# B&R Automation Studio project Mapp6D_Demo (part 2)

#### Variables.var - Local variables
```iecst
VAR
	DemoMacro : ARRAY[0..99] OF Macro_typ;
	gMacro : ARRAY[0..99] OF Macro_typ;
	MC_BR_MoveInPlaneAsync_Acp6D_0 : MC_BR_MoveInPlaneAsync_Acp6D;
	MC_BR_Move6D_Acp6D_0 : MC_BR_Move6D_Acp6D;
	MC_BR_MoveArc_Acp6D_0 : MC_BR_MoveArc_Acp6D;
	MC_BR_AsmPowerOn_Acp6D_0 : MC_BR_AsmPowerOn_Acp6D;
	MC_BR_MacroCreate_Acp6D_0 : MC_BR_MacroCreate_Acp6D;
	MC_BR_MoveInPlane_Acp6D_0 : MC_BR_MoveInPlane_Acp6D;
	MC_BR_AsmReadStatus_0 : MC_BR_AsmReadStatus_Acp6D;
	MC_BR_MacroSave_0 : MC_BR_MacroSave_Acp6D;
	MC_BR_MacroClear_0 : MC_BR_MacroClear_Acp6D;
	MC_BR_MacroDelete_0 : MC_BR_MacroDelete_Acp6D;
	MC_BR_MacroRun_0 : MC_BR_MacroRun_Acp6D;
	MC_BR_AsmGetShuttle_0 : MC_BR_AsmGetShuttle_Acp6D;
END_VAR
VAR CONSTANT
	MAX_NUM_SH : USINT := 10;
	C_MOVE_IN_PLANE_010 : USINT := 10;
	C_MOVE_IN_PLANE_ASYNC_015 : USINT := 15;
	C_MOVE_IN_6D_PLANE_020 : USINT := 20;
	C_MOVE_ARC_025 : USINT := 25;
	C_NEXT_COMMAND_05 : USINT := 5;
END_VAR
VAR
	Cmd : Ctrl_typ;
	i : USINT;
	inc : USINT;
	MacroState : USINT;
	visMacroStatus : STRING[80];
	MacroSh : {REDUND_UNREPLICABLE} ARRAY[0..9] OF Mc6DShuttleType;
	TempName : STRING[33];
	ExistingMacroNames : ARRAY[0..19] OF STRING[28];
	MacroName : STRING[28];
	helpStr : STRING[28];
	int_to_str : STRING[4];
	ShRefArr : ARRAY[0..MAX_NUM_SH] OF Mc6DShuttleType;
	macroLine : UDINT;
	command : UINT;
	Clear : BOOL;
	ReRun : BOOL;
	RunMacro : BOOL;
	CenterSegX : REAL;
	CenterSegY : REAL;
	SecondPosY : REAL;
	SecondPosX : REAL;
	FirstPosY : REAL;
	FirstPosX : REAL;
	visLockRun : BOOL;
	PathCW : McAcp6DInPlanePathEnum;
	PathACW : McAcp6DInPlanePathEnum;
END_VAR
VAR CONSTANT
	C_WAIT_00 : USINT := 0;
	C_READ_STATUS_01 : USINT := 1;
	C_POWER_ON_02 : USINT := 2;
	C_CREATE_03 : USINT := 3;
	C_DELETE_04 : USINT := 4;
	C_SAVE_60 : USINT := 60;
	C_REMAKE_DEMO_MACRO_70 : USINT := 70;
	C_RUN_DEMO_MACRO_80 : USINT := 80;
	C_RUN_DEMO_MACRO_81 : USINT := 81;
	C_RUN_DEMO_MACRO_82 : USINT := 82;
	C_RUN_DEMO_MACRO_83 : USINT := 83;
	C_RE_RUN_85 : USINT := 85;
	C_CLEARMACRO_90 : USINT := 90;
	C_RESET_100 : USINT := 100;
END_VAR
```

#### DemoAct.st
```iecst
ACTION DemoAct:

	// DEMO MACRO
	macroLine := 0;
	XY_MIN; 			// Min position on one segment 0.6 `
	XY_MAX; 			// Max position on one segment 0.240
	SEG_CENTER;			// Middle position 0.120

	// Calculate the min and max movement positions allowed

	IF inc = 0 THEN // System Top right 1st position
		FirstPosX := gAssemblyX_max;
		FirstPosY := gAssemblyY_max;
		SecondPosX := XY_MIN;
		SecondPosY := XY_MIN;
		CenterSegX := SEG_CENTER;
		CenterSegY := SEG_CENTER;
		PathCW := mcACP6D_PATH_Y_THEN_X;
		PathACW := mcACP6D_PATH_X_THEN_Y;
	ELSIF inc = 1 THEN // Bottom Left of system 1st position
		FirstPosX := XY_MIN;
		FirstPosY := XY_MIN;
		SecondPosX := gAssemblyX_max;
		SecondPosY := gAssemblyY_max;
		CenterSegX := gAssemblyX_max - HALF_SHUTTLE;
		CenterSegY := gAssemblyY_max - HALF_SHUTTLE;
		PathCW := mcACP6D_PATH_Y_THEN_X;
		PathACW := mcACP6D_PATH_X_THEN_Y;
	ELSIF inc = 2 THEN // Top left of system 1st position
		FirstPosX := XY_MIN;
		FirstPosY := gAssemblyY_max;
		SecondPosX := gAssemblyX_max;
		SecondPosY := XY_MIN;
		CenterSegX := gAssemblyX_max - HALF_SHUTTLE;
		CenterSegY := SEG_CENTER;
		PathCW := mcACP6D_PATH_X_THEN_Y;
		PathACW := mcACP6D_PATH_Y_THEN_X;
	ELSIF inc = 3 THEN // Bottom right of system 1st position
		FirstPosX := gAssemblyX_max;
		FirstPosY := XY_MIN;
		SecondPosX := XY_MIN;
		SecondPosY := gAssemblyY_max;
		CenterSegX := SEG_CENTER;
		CenterSegY := gAssemblyY_max - HALF_SHUTTLE;
		PathCW := mcACP6D_PATH_X_THEN_Y;
		PathACW := mcACP6D_PATH_Y_THEN_X;
	END_IF

	// Round edge twice total CWise

	DemoMacro[macroLine].ShuttleID := 1;
	DemoMacro[macroLine].CommandType := C_MOVE_IN_PLANE_010;
	DemoMacro[macroLine].MovePlane.Velocity := 2.0;
	DemoMacro[macroLine].MovePlane.Acceleration := 20.0;
	DemoMacro[macroLine].MovePlane.EndVelocity := 0.0;
	DemoMacro[macroLine].MovePlane.Position.X := FirstPosX;
	DemoMacro[macroLine].MovePlane.Position.Y := FirstPosY;
	DemoMacro[macroLine].MovePlane.Path := PathCW;

	macroLine := macroLine + 1;

	DemoMacro[macroLine].ShuttleID := 1;
	DemoMacro[macroLine].CommandType := C_MOVE_IN_PLANE_010;
	DemoMacro[macroLine].MovePlane.Velocity := 2.0;
	DemoMacro[macroLine].MovePlane.Acceleration := 20.0;
	DemoMacro[macroLine].MovePlane.EndVelocity := 0.0;
	DemoMacro[macroLine].MovePlane.Position.X := SecondPosX;
	DemoMacro[macroLine].MovePlane.Position.Y := SecondPosY;
	DemoMacro[macroLine].MovePlane.Path := PathCW;

	macroLine := macroLine + 1;

	DemoMacro[macroLine].ShuttleID := 1;
	DemoMacro[macroLine].CommandType := C_MOVE_IN_PLANE_010;
	DemoMacro[macroLine].MovePlane.Velocity := 2.0;
	DemoMacro[macroLine].MovePlane.Acceleration := 20.0;
	DemoMacro[macroLine].MovePlane.EndVelocity := 0.0;
	DemoMacro[macroLine].MovePlane.Position.X := FirstPosX;
	DemoMacro[macroLine].MovePlane.Position.Y := FirstPosY;
	DemoMacro[macroLine].MovePlane.Path := PathCW;

	macroLine := macroLine + 1;

	DemoMacro[macroLine].ShuttleID := 1;
	DemoMacro[macroLine].CommandType := C_MOVE_IN_PLANE_010;
	DemoMacro[macroLine].MovePlane.Velocity := 2.0;
	DemoMacro[macroLine].MovePlane.Acceleration := 20.0;
	DemoMacro[macroLine].MovePlane.EndVelocity := 0.0;
	DemoMacro[macroLine].MovePlane.Position.X := SecondPosX;
	DemoMacro[macroLine].MovePlane.Position.Y := SecondPosY;
	DemoMacro[macroLine].MovePlane.Path := PathCW;

	macroLine := macroLine + 1;

	// Move to center and dance...
	DemoMacro[macroLine].ShuttleID 					  := 1;
	DemoMacro[macroLine].CommandType 				  := C_MOVE_IN_6D_PLANE_020;
	DemoMacro[macroLine].Move6D.ShortAxis.Velocity.Z  := 0.1;
	DemoMacro[macroLine].Move6D.ShortAxis.Position.Z  := 0.003;
	DemoMacro[macroLine].Move6D.ShortAxis.Velocity.Rz := 0.3;
	DemoMacro[macroLine].Move6D.ShortAxis.Position.Rz := 0.086;
	DemoMacro[macroLine].Move6D.ShortAxis.Velocity.Rx := 0.1;
	DemoMacro[macroLine].Move6D.ShortAxis.Position.Rx := -0.015;
	DemoMacro[macroLine].Move6D.ShortAxis.Velocity.Ry := 0.1;
	DemoMacro[macroLine].Move6D.ShortAxis.Position.Ry := -0.015;
	DemoMacro[macroLine].Move6D.InPlane.Velocity      := 0.2;
	DemoMacro[macroLine].Move6D.InPlane.Acceleration  := 10;
	DemoMacro[macroLine].Move6D.InPlane.Position.X    := CenterSegX;
	DemoMacro[macroLine].Move6D.InPlane.Position.Y    := CenterSegY;

	macroLine := macroLine + 1;

	DemoMacro[macroLine].ShuttleID 					  := 1;
	DemoMacro[macroLine].CommandType 				  := C_MOVE_IN_6D_PLANE_020;
	DemoMacro[macroLine].Move6D.ShortAxis.Velocity.Z  := 0.1;
	DemoMacro[macroLine].Move6D.ShortAxis.Position.Z  := 0.001;
	DemoMacro[macroLine].Move6D.ShortAxis.Velocity.Rz := 0.3;
	DemoMacro[macroLine].Move6D.ShortAxis.Position.Rz := -0.086;
	DemoMacro[macroLine].Move6D.ShortAxis.Velocity.Rx := 0.1;
	DemoMacro[macroLine].Move6D.ShortAxis.Position.Rx := 0.00;
	DemoMacro[macroLine].Move6D.ShortAxis.Velocity.Ry := 0.1;
	DemoMacro[macroLine].Move6D.ShortAxis.Position.Ry := 0.00;
	DemoMacro[macroLine].Move6D.InPlane.Velocity      := 0.2;
	DemoMacro[macroLine].Move6D.InPlane.Acceleration  := 10;
	DemoMacro[macroLine].Move6D.InPlane.Position.X    := CenterSegX;
	DemoMacro[macroLine].Move6D.InPlane.Position.Y    := CenterSegY;

	macroLine := macroLine + 1;

	DemoMacro[macroLine].ShuttleID 					  := 1;
	DemoMacro[macroLine].CommandType 				  := C_MOVE_IN_6D_PLANE_020;
	DemoMacro[macroLine].Move6D.ShortAxis.Velocity.Z  := 0.1;
	DemoMacro[macroLine].Move6D.ShortAxis.Position.Z  := 0.004;
	DemoMacro[macroLine].Move6D.ShortAxis.Velocity.Rz := 0.3;
	DemoMacro[macroLine].Move6D.ShortAxis.Position.Rz := 0.0;
	DemoMacro[macroLine].Move6D.ShortAxis.Velocity.Rx := 0.1;
	DemoMacro[macroLine].Move6D.ShortAxis.Position.Rx := -0.015;
	DemoMacro[macroLine].Move6D.ShortAxis.Velocity.Ry := 0.1;
	DemoMacro[macroLine].Move6D.ShortAxis.Position.Ry := -0.015;
	DemoMacro[macroLine].Move6D.InPlane.Velocity      := 0.2;
	DemoMacro[macroLine].Move6D.InPlane.Acceleration  := 10;
	DemoMacro[macroLine].Move6D.InPlane.Position.X    := CenterSegX;
	DemoMacro[macroLine].Move6D.InPlane.Position.Y    := CenterSegY;

	macroLine := macroLine + 1;

	DemoMacro[macroLine].ShuttleID 					  := 1;
	DemoMacro[macroLine].CommandType 				  := C_MOVE_IN_6D_PLANE_020;
	DemoMacro[macroLine].Move6D.ShortAxis.Velocity.Z  := 0.1;
	DemoMacro[macroLine].Move6D.ShortAxis.Position.Z  := 0.004;
	DemoMacro[macroLine].Move6D.ShortAxis.Velocity.Rz := 0.3;
	DemoMacro[macroLine].Move6D.ShortAxis.Position.Rz := 0.0;
	DemoMacro[macroLine].Move6D.ShortAxis.Velocity.Rx := 0.1;
	DemoMacro[macroLine].Move6D.ShortAxis.Position.Rx := -0.015;
	DemoMacro[macroLine].Move6D.ShortAxis.Velocity.Ry := 0.1;
	DemoMacro[macroLine].Move6D.ShortAxis.Position.Ry := 0;
	DemoMacro[macroLine].Move6D.InPlane.Velocity      := 0.2;
	DemoMacro[macroLine].Move6D.InPlane.Acceleration  := 10;
	DemoMacro[macroLine].Move6D.InPlane.Position.X    := CenterSegX;
	DemoMacro[macroLine].Move6D.InPlane.Position.Y    := CenterSegY;

	macroLine := macroLine + 1;

	DemoMacro[macroLine].ShuttleID 					  := 1;
	DemoMacro[macroLine].CommandType 				  := C_MOVE_IN_6D_PLANE_020;
	DemoMacro[macroLine].Move6D.ShortAxis.Velocity.Z  := 0.1;
	DemoMacro[macroLine].Move6D.ShortAxis.Position.Z  := 0.004;
	DemoMacro[macroLine].Move6D.ShortAxis.Velocity.Rz := 0.3;
	DemoMacro[macroLine].Move6D.ShortAxis.Position.Rz := 0.0;
	DemoMacro[macroLine].Move6D.ShortAxis.Velocity.Rx := 0.1;
	DemoMacro[macroLine].Move6D.ShortAxis.Position.Rx := 0;
	DemoMacro[macroLine].Move6D.ShortAxis.Velocity.Ry := 0.1;
	DemoMacro[macroLine].Move6D.ShortAxis.Position.Ry := 0.015;
	DemoMacro[macroLine].Move6D.InPlane.Velocity      := 0.2;
	DemoMacro[macroLine].Move6D.InPlane.Acceleration  := 10;
	DemoMacro[macroLine].Move6D.InPlane.Position.X    := CenterSegX;
	DemoMacro[macroLine].Move6D.InPlane.Position.Y    := CenterSegY;

	macroLine := macroLine + 1;

	DemoMacro[macroLine].ShuttleID 					  := 1;
	DemoMacro[macroLine].CommandType 				  := C_MOVE_IN_6D_PLANE_020;
	DemoMacro[macroLine].Move6D.ShortAxis.Velocity.Z  := 0.1;
	DemoMacro[macroLine].Move6D.ShortAxis.Position.Z  := 0.004;
	DemoMacro[macroLine].Move6D.ShortAxis.Velocity.Rz := 0.3;
	DemoMacro[macroLine].Move6D.ShortAxis.Position.Rz := 0.0;
	DemoMacro[macroLine].Move6D.ShortAxis.Velocity.Rx := 0.1;
	DemoMacro[macroLine].Move6D.ShortAxis.Position.Rx := 0.015;
	DemoMacro[macroLine].Move6D.ShortAxis.Velocity.Ry := 0.1;
	DemoMacro[macroLine].Move6D.ShortAxis.Position.Ry := 0.015;
	DemoMacro[macroLine].Move6D.InPlane.Velocity      := 0.2;
	DemoMacro[macroLine].Move6D.InPlane.Acceleration  := 10;
	DemoMacro[macroLine].Move6D.InPlane.Position.X    := CenterSegX;
	DemoMacro[macroLine].Move6D.InPlane.Position.Y    := CenterSegY;

	macroLine := macroLine + 1;

	DemoMacro[macroLine].ShuttleID 					  := 1;
	DemoMacro[macroLine].CommandType 				  := C_MOVE_IN_6D_PLANE_020;
	DemoMacro[macroLine].Move6D.ShortAxis.Velocity.Z  := 0.1;
	DemoMacro[macroLine].Move6D.ShortAxis.Position.Z  := 0.004;
	DemoMacro[macroLine].Move6D.ShortAxis.Velocity.Rz := 0.3;
	DemoMacro[macroLine].Move6D.ShortAxis.Position.Rz := 0.0;
	DemoMacro[macroLine].Move6D.ShortAxis.Velocity.Rx := 0.1;
	DemoMacro[macroLine].Move6D.ShortAxis.Position.Rx := 0.015;
	DemoMacro[macroLine].Move6D.ShortAxis.Velocity.Ry := 0.1;
	DemoMacro[macroLine].Move6D.ShortAxis.Position.Ry := 0;
	DemoMacro[macroLine].Move6D.InPlane.Velocity      := 0.2;
	DemoMacro[macroLine].Move6D.InPlane.Acceleration  := 10;
	DemoMacro[macroLine].Move6D.InPlane.Position.X    := CenterSegX;
	DemoMacro[macroLine].Move6D.InPlane.Position.Y    := CenterSegY;

	macroLine := macroLine + 1;

	DemoMacro[macroLine].ShuttleID 					  := 1;
	DemoMacro[macroLine].CommandType 				  := C_MOVE_IN_6D_PLANE_020;
	DemoMacro[macroLine].Move6D.ShortAxis.Velocity.Z  := 0.1;
	DemoMacro[macroLine].Move6D.ShortAxis.Position.Z  := 0.004;
	DemoMacro[macroLine].Move6D.ShortAxis.Velocity.Rz := 0.3;
	DemoMacro[macroLine].Move6D.ShortAxis.Position.Rz := 0.0;
	DemoMacro[macroLine].Move6D.ShortAxis.Velocity.Rx := 0.1;
	DemoMacro[macroLine].Move6D.ShortAxis.Position.Rx := 0.0;
	DemoMacro[macroLine].Move6D.ShortAxis.Velocity.Ry := 0.1;
	DemoMacro[macroLine].Move6D.ShortAxis.Position.Ry := -0.015;
	DemoMacro[macroLine].Move6D.InPlane.Velocity      := 0.2;
	DemoMacro[macroLine].Move6D.InPlane.Acceleration  := 10;
	DemoMacro[macroLine].Move6D.InPlane.Position.X    := CenterSegX;
	DemoMacro[macroLine].Move6D.InPlane.Position.Y    := CenterSegY;

	macroLine := macroLine + 1;

	DemoMacro[macroLine].ShuttleID 					  := 1;
	DemoMacro[macroLine].CommandType 				  := C_MOVE_IN_6D_PLANE_020;
	DemoMacro[macroLine].Move6D.ShortAxis.Velocity.Z  := 0.1;
	DemoMacro[macroLine].Move6D.ShortAxis.Position.Z  := 0.004;
	DemoMacro[macroLine].Move6D.ShortAxis.Velocity.Rz := 0.3;
	DemoMacro[macroLine].Move6D.ShortAxis.Position.Rz := 0.0;
	DemoMacro[macroLine].Move6D.ShortAxis.Velocity.Rx := 0.1;
	DemoMacro[macroLine].Move6D.ShortAxis.Position.Rx := -0.015;
	DemoMacro[macroLine].Move6D.ShortAxis.Velocity.Ry := 0.1;
	DemoMacro[macroLine].Move6D.ShortAxis.Position.Ry := -0.015;
	DemoMacro[macroLine].Move6D.InPlane.Velocity      := 0.2;
	DemoMacro[macroLine].Move6D.InPlane.Acceleration  := 10;
	DemoMacro[macroLine].Move6D.InPlane.Position.X    := CenterSegX;
	DemoMacro[macroLine].Move6D.InPlane.Position.Y    := CenterSegY;

	macroLine := macroLine + 1;

	// RESET Short Axes
	DemoMacro[macroLine].ShuttleID 					  := 1;
	DemoMacro[macroLine].CommandType 				  := C_MOVE_IN_6D_PLANE_020;
	DemoMacro[macroLine].Move6D.ShortAxis.Velocity.Z  := 0.1;
	DemoMacro[macroLine].Move6D.ShortAxis.Position.Z  := 0.001;
	DemoMacro[macroLine].Move6D.ShortAxis.Velocity.Rz := 0.3;
	DemoMacro[macroLine].Move6D.ShortAxis.Position.Rz := 0.0;
	DemoMacro[macroLine].Move6D.ShortAxis.Velocity.Rx := 0.1;
	DemoMacro[macroLine].Move6D.ShortAxis.Position.Rx := 0.0;
	DemoMacro[macroLine].Move6D.ShortAxis.Velocity.Ry := 0.1;
	DemoMacro[macroLine].Move6D.ShortAxis.Position.Ry := 0.0;
	DemoMacro[macroLine].Move6D.InPlane.Velocity      := 0.2;
	DemoMacro[macroLine].Move6D.InPlane.Acceleration  := 10;
	DemoMacro[macroLine].Move6D.InPlane.Position.X    := CenterSegX;
	DemoMacro[macroLine].Move6D.InPlane.Position.Y    := CenterSegY;

	macroLine := macroLine + 1;

	// Round edge twice total ACWise

	DemoMacro[macroLine].ShuttleID := 1;
	DemoMacro[macroLine].CommandType := C_MOVE_IN_PLANE_010;
	DemoMacro[macroLine].MovePlane.Velocity := 2.0;
	DemoMacro[macroLine].MovePlane.Acceleration := 20.0;
	DemoMacro[macroLine].MovePlane.EndVelocity := 0.0;
	DemoMacro[macroLine].MovePlane.Position.X := SecondPosX;
	DemoMacro[macroLine].MovePlane.Position.Y := SecondPosY;
	DemoMacro[macroLine].MovePlane.Path := PathACW;

	macroLine := macroLine + 1;

	DemoMacro[macroLine].ShuttleID := 1;
	DemoMacro[macroLine].CommandType := C_MOVE_IN_PLANE_010;
	DemoMacro[macroLine].MovePlane.Velocity := 2.0;
	DemoMacro[macroLine].MovePlane.Acceleration := 20.0;
	DemoMacro[macroLine].MovePlane.EndVelocity := 0.0;
	DemoMacro[macroLine].MovePlane.Position.X := FirstPosX;
	DemoMacro[macroLine].MovePlane.Position.Y := FirstPosY;
	DemoMacro[macroLine].MovePlane.Path := PathACW;

	macroLine := macroLine + 1;

	DemoMacro[macroLine].ShuttleID := 1;
	DemoMacro[macroLine].CommandType := C_MOVE_IN_PLANE_010;
	DemoMacro[macroLine].MovePlane.Velocity := 2.0;
	DemoMacro[macroLine].MovePlane.Acceleration := 20.0;
	DemoMacro[macroLine].MovePlane.EndVelocity := 0.0;
	DemoMacro[macroLine].MovePlane.Position.X := SecondPosX;
	DemoMacro[macroLine].MovePlane.Position.Y := SecondPosY;
	DemoMacro[macroLine].MovePlane.Path := PathACW;

	macroLine := macroLine + 1;

	DemoMacro[macroLine].ShuttleID := 1;
	DemoMacro[macroLine].CommandType := C_MOVE_IN_PLANE_010;
	DemoMacro[macroLine].MovePlane.Velocity := 2.0;
	DemoMacro[macroLine].MovePlane.Acceleration := 20.0;
	DemoMacro[macroLine].MovePlane.EndVelocity := 0.0;
	DemoMacro[macroLine].MovePlane.Position.X := FirstPosX;
	DemoMacro[macroLine].MovePlane.Position.Y := FirstPosY;
	DemoMacro[macroLine].MovePlane.Path := PathACW;

	macroLine := macroLine + 1;

	DemoMacro[macroLine].ShuttleID := 1;
	DemoMacro[macroLine].CommandType := 60;
	gMacro := DemoMacro;

END_ACTION
```

### Program Logical/ShuttleGroup (IEC)

#### Variables.var
```iecst
VAR
	MC_BR_ShGroupCreate_0 : MC_BR_ShGroupCreate_Acp6D;
	MC_BR_AsmPowerOn_Acp6D_0 : MC_BR_AsmPowerOn_Acp6D;
	MC_BR_AsmReadStatus_0 : MC_BR_AsmReadStatus_Acp6D;
	Cmd : Ctrl_typ;
	ShGroupState : USINT;
	ShGroupRef : Mc6DShuttleGroupType;
	MC_BR_ShGroupAddShuttle_0 : MC_BR_ShGroupAddShuttle_Acp6D;
	MC_BR_AsmGetShuttle_0 : MC_BR_AsmGetShuttle_Acp6D;
	ShRefArr : ARRAY[0..MAX_NUM_SH] OF Mc6DShuttleType;
END_VAR
VAR CONSTANT
	MAX_NUM_SH : USINT := 10;
END_VAR
VAR
	i : USINT;
	MC_BR_ShGroupClear_0 : MC_BR_ShGroupClear_Acp6D;
	MC_BR_ShGroupGetInfo_0 : MC_BR_ShGroupGetInfo_Acp6D;
	MC_BR_ShGroupCoupleCtrl_0 : MC_BR_ShGroupCoupleCtrl_Acp6D;
	MC_BR_ShGroupBuffer_0 : MC_BR_ShGroupBuffer_Acp6D;
	MC_BR_AsmGetShGroup_0 : MC_BR_AsmGetShGroup_Acp6D;
	MC_BR_ShGroupDelete_0 : MC_BR_ShGroupDelete_Acp6D;
END_VAR
```

### Program Logical/VirtualShuttle1 (IEC)

#### Variables.var
```iecst
VAR
	MC_BR_ShGroupCreate_0 : MC_BR_ShGroupCreate_Acp6D;
	MC_BR_AsmPowerOn_Acp6D_0 : MC_BR_AsmPowerOn_Acp6D;
	MC_BR_AsmReadStatus_0 : MC_BR_AsmReadStatus_Acp6D;
	Cmd : Ctrl_typ;
	VirtualShState : USINT;
	VirtualShRef : Mc6DShuttleGroupType;
	MC_BR_ShGroupAddShuttle_0 : MC_BR_ShGroupAddShuttle_Acp6D;
	MC_BR_AsmGetShuttle_0 : MC_BR_AsmGetShuttle_Acp6D;
	VirtualShRefArr : ARRAY[0..MAX_NUM_SH] OF Mc6DShuttleType;
END_VAR
VAR CONSTANT
	MAX_NUM_SH : USINT := 10;
END_VAR
VAR
	i : USINT;
	MC_BR_AsmGetVirtualSh_0 : MC_BR_AsmGetVirtualSh_Acp6D;
	MC_BR_VirtualShCreate_0 : MC_BR_VirtualShCreate_Acp6D;
	MC_BR_MoveInPlane_0 : MC_BR_MoveInPlane_Acp6D;
END_VAR
```

### Program Logical/Planet (IEC)

#### Variables.var
```iecst
VAR
	MC_BR_ShGroupCreate_0 : MC_BR_ShGroupCreate_Acp6D;
	MC_BR_AsmPowerOn_Acp6D_0 : MC_BR_AsmPowerOn_Acp6D;
	MC_BR_AsmReadStatus_0 : MC_BR_AsmReadStatus_Acp6D;
	Cmd : Ctrl_typ;
	PlanetState : USINT;
	VirtualShRef : Mc6DShuttleGroupType;
	MC_BR_AsmGetShuttle_0 : MC_BR_AsmGetShuttle_Acp6D;
	PlanetShRefArr : ARRAY[0..MAX_NUM_SH] OF Mc6DShuttleType;
END_VAR
VAR CONSTANT
	MAX_NUM_SH : USINT := 10;
END_VAR
VAR
	i : USINT;
	MC_BR_VirtualShCreate_0 : MC_BR_VirtualShCreate_Acp6D;
	MC_BR_AsmGetVirtualSh_0 : MC_BR_AsmGetVirtualSh_Acp6D;
	MC_BR_MoveInPlane_0 : MC_BR_MoveInPlane_Acp6D;
	MC_BR_ShPlanet_0 : MC_BR_ShPlanet_Acp6D;
END_VAR
```

- Visualisation Logical/mappView (not shown)

### Program Logical/HMI (IEC)

#### Types.typ
```iecst
TYPE
	workStationList_typ : 	STRUCT
		listProvider : STRING[800];
		stationCounter : USINT;
		tmpString : STRING[80];
	END_STRUCT;
	local_typ : 	STRUCT
		workStationList : workStationList_typ;
		tableConfigClick : BOOL;
		tableConfigString : STRING[80];
		tableConfigID : USINT;
	END_STRUCT;
END_TYPE
```

#### Variables.var
```iecst
VAR
	visSelectedShuttle : STRING[10];
	demoMotorSegmentLayoutCmd : BOOL;
	i : USINT;
	init : BOOL;
	j : INT;
	nrOfShuttlesHMI : USINT := 15;
	pSegments : REFERENCE TO MotorSegments_typ;
	pShuttleInfo : REFERENCE TO ShuttleInfo_typ;
	pShuttleStartupInfo : REFERENCE TO ShuttleStartup_typ;
	resetMotorSegmentLayoutCmd : BOOL;
	resetShuttleInitLayoutCmd : BOOL;
	showConfigShuttles : STRING[5000];
	showConfigSvg : BOOL := TRUE;
	showConfigSvgCmd : BOOL;
	showShuttlesPosRx : STRING[1000];
	showShuttlesPosRy : STRING[1000];
	showShuttles : STRING[5000];
	showTyleSvg : BOOL;
	showTyleSvgCmd : BOOL;
	shuttleStartPosSvg : BOOL;
	shuttleStartPosSvgCmd : BOOL;
	sizeOfArray2 : DINT;
	sizeOfArray1 : DINT;
	sizeOfArray : DINT;
	this : local_typ;
	tmpCalc : REAL;
	tmpString : STRING[5000];
	xCordinate : INT;
	yCordinate : INT;
	testValue : REAL;
	TESTString : STRING[2000];
	TempTestString : STRING[10];
	XOffset : REAL;
	YOffset : REAL;
	MTLookUpTable_0 : MTLookUpTable;
	offsetOut : ARRAY[0..49] OF REAL;
	offsetHeight : ARRAY[0..49] OF REAL;
END_VAR
```

#### drawConfigShuttles.st
```iecst
ACTION drawConfigShuttles:
	IF shuttleStartPosSvg OR init THEN
		IF i = 0 THEN
		showConfigShuttles := '';
		tmpString := gShowMotorSegments;
		brdkStrRemove(ADR(tmpString),-1,1);
		brdkStrCat(ADR(showConfigShuttles), ADR(tmpString));
		brdkStrCat(ADR(showConfigShuttles), ADR(','));
		END_IF

		brdkStrCat(ADR(showConfigShuttles), ADR('{"select":"#rect'));

		tmpString := USINT_TO_STRING(i+1);
		brdkStrCat(ADR(showConfigShuttles), ADR(tmpString));
		brdkStrCat(ADR(showConfigShuttles), ADR('","display":'));
		IF (nrOfShuttlesHMI >= (i+1)) THEN
			brdkStrCat(ADR(showConfigShuttles), ADR('true'));
		ELSE
			brdkStrCat(ADR(showConfigShuttles), ADR('false'));
		END_IF

		brdkStrCat(ADR(showConfigShuttles), ADR(',"translate":['));

		tmpCalc := (pShuttleStartupInfo.initXPos*1000)-60;
		tmpString := REAL_TO_STRING(tmpCalc);
		brdkStrCat(ADR(showConfigShuttles), ADR(tmpString));
		brdkStrCat(ADR(showConfigShuttles), ADR(','));

		tmpCalc := 1200 - (pShuttleStartupInfo.initYPos*1000) - 60;
		tmpString := REAL_TO_STRING(tmpCalc);
		brdkStrCat(ADR(showConfigShuttles), ADR(tmpString));

		IF i = MAX_NUM_SHUTTLES THEN
			brdkStrCat(ADR(showConfigShuttles), ADR(']}]'));
		ELSE
			brdkStrCat(ADR(showConfigShuttles), ADR(']},'));
		END_IF

		//	brdkStrCat(ADR(showConfigShuttles), ADR('<text x="50%" y="50%" dominant-baseline="middle" text-anchor="middle">weight</text>'));

	END_IF

END_ACTION
```

#### drawMotorSegments.st
```iecst
ACTION drawMotorSegments:
	IF showTyleSvg OR init THEN
		IF i = 0 THEN
			gShowMotorSegments := '';
			brdkStrCat(ADR(gShowMotorSegments), ADR('[{"select":"#MS'));
		ELSE
			brdkStrCat(ADR(gShowMotorSegments), ADR('{"select":"#MS'));
		END_IF

		tmpString := USINT_TO_STRING(i+1);
		brdkStrCat(ADR(gShowMotorSegments), ADR(tmpString));
		brdkStrCat(ADR(gShowMotorSegments), ADR('","display":'));
		IF pSegments.visible THEN
			brdkStrCat(ADR(gShowMotorSegments), ADR('true'));
		ELSE
			brdkStrCat(ADR(gShowMotorSegments), ADR('false'));
		END_IF

		IF i = NR_OF_SEGMENTS THEN
			brdkStrCat(ADR(gShowMotorSegments), ADR('}]'));
		ELSE
			brdkStrCat(ADR(gShowMotorSegments), ADR('},'));
		END_IF
	END_IF

	IF i = NR_OF_SEGMENTS THEN
		showTyleSvg := FALSE;
		init := FALSE;
	END_IF

END_ACTION
```

#### drawShuttles.st
```iecst
ACTION drawShuttles:

		//////////// CREATE TEXT CODE /////////
	// Create the Texts
	IF (i < gMain.Status.ShuttlesPresent) AND (gMain.Status.Ready) THEN
		IF i = 0 THEN
			TESTString := '';
		END_IF

		IF pShuttleInfo.State <> mcACP6D_SH_STATE_MOTION THEN
		brdkStrCat(ADR(TESTString), ADR('<text class="ShtId'));
		TempTestString := UINT_TO_STRING(gShuttleReference[i].ID);
		brdkStrCat(ADR(TESTString), ADR(TempTestString));
		brdkStrCat(ADR(TESTString), ADR('" font-family="Helvetica, Arial, sans-serif" font-size="25" y="'));

		MTLookUpTable_0.Enable := TRUE;
		MTLookUpTable_0.InX := pShuttleInfo.Position.Y;
		MTLookUpTable_0();
		YOffset := MTLookUpTable_0.Out;
		// Add Y position
		tmpCalc := YOffset-((pShuttleInfo.Position.Y));
		TempTestString := REAL_TO_STRING(tmpCalc);
		brdkStrCat(ADR(TESTString), ADR(TempTestString));

		// ADD X position
		brdkStrCat(ADR(TESTString), ADR('" x="'));
		tmpCalc := ((pShuttleInfo.Position.X));// * 2)) - XOffset;

		TempTestString := REAL_TO_STRING(tmpCalc);
		brdkStrCat(ADR(TESTString), ADR(TempTestString));

		// Add the Text
		brdkStrCat(ADR(TESTString), ADR('">ID:'));
		TempTestString := USINT_TO_STRING(pShuttleInfo.ID);
		brdkStrCat(ADR(TESTString), ADR(TempTestString));
			brdkStrCat(ADR(TESTString), ADR('</text>'));
		ELSE

		END_IF

	END_IF
	///////

	// Change the rectangles //
	IF i = 0 THEN
		showShuttles := '';
		tmpString := gShowMotorSegments;
		brdkStrRemove(ADR(tmpString),-1,1);
		brdkStrCat(ADR(showShuttles), ADR(tmpString));
		brdkStrCat(ADR(showShuttles), ADR(','));
	END_IF

	brdkStrCat(ADR(showShuttles), ADR('{"select":"#rect'));

	tmpString := USINT_TO_STRING(i+1);
	brdkStrCat(ADR(showShuttles), ADR(tmpString));
	brdkStrCat(ADR(showShuttles), ADR('","display":'));
	IF (nrOfShuttlesHMI >= (i+1))AND(pShuttleInfo.State <> mcACP6D_SH_STATE_RESERVED)THEN
		brdkStrCat(ADR(showShuttles), ADR('true'));
	ELSE
		brdkStrCat(ADR(showShuttles), ADR('false'));
	END_IF

	IF(pShuttleInfo.State = mcACP6D_SH_STATE_OBSTACLE)THEN
		brdkStrCat(ADR(showShuttles), ADR(',"style":"fill:4;')); // Yellow
	ELSIF(pShuttleInfo.State = mcACP6D_SH_STATE_STOPPED)THEN // RED
		brdkStrCat(ADR(showShuttles), ADR(',"style":"fill:0;'));
	ELSIF pShuttleInfo.State = mcACP6D_SH_STATE_LANDED THEN // BLUE
		brdkStrCat(ADR(showShuttles), ADR(',"style":"fill:2;'));
	ELSIF pShuttleInfo.State = mcACP6D_SH_STATE_DISABLED THEN // Red/maroon
		brdkStrCat(ADR(showShuttles), ADR(',"style":"fill:3;'));
	ELSE									// Black border white
		brdkStrCat(ADR(showShuttles), ADR(',"style":"fill:6;'));
	END_IF

	IF (gMain.Par.SelectedIndex = i)THEN // Green border
	brdkStrCat(ADR(showShuttles), ADR('stroke:5;stroke-width:5px;"'));
	ELSE								// Black border
	brdkStrCat(ADR(showShuttles), ADR('stroke:7;stroke-width:1px;"'));
	END_IF

	brdkStrCat(ADR(showShuttles), ADR(',"translate":['));

	tmpCalc := ((pShuttleInfo.Position.X * 2))-120;
	tmpString := REAL_TO_STRING(tmpCalc);
	brdkStrCat(ADR(showShuttles), ADR(tmpString));
	brdkStrCat(ADR(showShuttles), ADR(','));

	tmpCalc := 960 - ((pShuttleInfo.Position.Y * 2))-120;
	tmpString := REAL_TO_STRING(tmpCalc);
	brdkStrCat(ADR(showShuttles), ADR(tmpString));

	brdkStrCat(ADR(showShuttles), ADR(']'));

	brdkStrCat(ADR(showShuttles), ADR(',"spin":['));

	tmpCalc := ((pShuttleInfo.Position.Rz/17.453293)*-1);
	tmpString := REAL_TO_STRING(tmpCalc);
	brdkStrCat(ADR(showShuttles), ADR(tmpString));
	brdkStrCat(ADR(showShuttles), ADR(',120,120'));
	// END Rectangles
//	brdkStrCat(ADR(showShuttles), ADR(']}'));

//	IF i = UINT_TO_USINT(gMain.Status.ShuttlesPresent)THEN
	IF i = 4 THEN
		brdkStrCat(ADR(showShuttles), ADR(']}]'));
	ELSE
		brdkStrCat(ADR(showShuttles), ADR(']},'));
	END_IF

	sizeOfArray := brdkStrLen(ADR(showShuttles));

	////////////////////////////////////////////////////////////////////////////////////
	////////////////////////////////////////////////////////////////////////////////////

	IF i = gMain.Par.SelectedIndex THEN

		// Display the Shuttle Rx position
		showShuttlesPosRx := '';
		brdkStrCat(ADR(showShuttlesPosRx), ADR('[{"select":"#ShuttleMain'));
		brdkStrCat(ADR(showShuttlesPosRx), ADR('","display":'));
		brdkStrCat(ADR(showShuttlesPosRx), ADR('true'));
		brdkStrCat(ADR(showShuttlesPosRx), ADR(',"translate":['));
		tmpCalc := (0);
		tmpString := REAL_TO_STRING(tmpCalc);
		brdkStrCat(ADR(showShuttlesPosRx), ADR(tmpString));
		brdkStrCat(ADR(showShuttlesPosRx), ADR(','));
		tmpCalc := (((pShuttleInfo.Position.Z)*-1)*5);
		tmpString := REAL_TO_STRING(tmpCalc);
		brdkStrCat(ADR(showShuttlesPosRx), ADR(tmpString));
		brdkStrCat(ADR(showShuttlesPosRx), ADR(']'));
		brdkStrCat(ADR(showShuttlesPosRx), ADR(',"spin":['));
		tmpCalc := ((pShuttleInfo.Position.Rx/17.453293));
		tmpString := REAL_TO_STRING(tmpCalc);
		brdkStrCat(ADR(showShuttlesPosRx), ADR(tmpString));
		brdkStrCat(ADR(showShuttlesPosRx), ADR(',200,2.5'));
		brdkStrCat(ADR(showShuttlesPosRx), ADR(']},'));
		brdkStrCat(ADR(showShuttlesPosRx), ADR('{"select":"#ShuttleTop'));
		brdkStrCat(ADR(showShuttlesPosRx), ADR('","display":'));
		brdkStrCat(ADR(showShuttlesPosRx), ADR('true'));
		brdkStrCat(ADR(showShuttlesPosRx), ADR(',"translate":['));
		tmpCalc := (0);
		tmpString := REAL_TO_STRING(tmpCalc);
		brdkStrCat(ADR(showShuttlesPosRx), ADR(tmpString));
		brdkStrCat(ADR(showShuttlesPosRx), ADR(','));
		tmpCalc := (((pShuttleInfo.Position.Z)*-1)*5);
		tmpString := REAL_TO_STRING(tmpCalc);
		brdkStrCat(ADR(showShuttlesPosRx), ADR(tmpString));
		brdkStrCat(ADR(showShuttlesPosRx), ADR(']'));
		brdkStrCat(ADR(showShuttlesPosRx), ADR(',"spin":['));
		tmpCalc := ((pShuttleInfo.Position.Rx/17.453293));
		tmpString := REAL_TO_STRING(tmpCalc);
		brdkStrCat(ADR(showShuttlesPosRx), ADR(tmpString));
		brdkStrCat(ADR(showShuttlesPosRx), ADR(',200,2.5'));
		brdkStrCat(ADR(showShuttlesPosRx), ADR(']}]'));
		sizeOfArray1 := brdkStrLen(ADR(showShuttlesPosRx));

		// Display the Shuttle Ry position
		showShuttlesPosRy := '';
		brdkStrCat(ADR(showShuttlesPosRy), ADR('[{"select":"#ShuttleMain'));
		brdkStrCat(ADR(showShuttlesPosRy), ADR('","display":'));
		brdkStrCat(ADR(showShuttlesPosRy), ADR('true'));
		brdkStrCat(ADR(showShuttlesPosRy), ADR(',"translate":['));
		tmpCalc := (0);
		tmpString := REAL_TO_STRING(tmpCalc);
		brdkStrCat(ADR(showShuttlesPosRy), ADR(tmpString));
		brdkStrCat(ADR(showShuttlesPosRy), ADR(','));
		tmpCalc := (((pShuttleInfo.Position.Z)*-1)*5);
		tmpString := REAL_TO_STRING(tmpCalc);
		brdkStrCat(ADR(showShuttlesPosRy), ADR(tmpString));
		brdkStrCat(ADR(showShuttlesPosRy), ADR(']'));
		brdkStrCat(ADR(showShuttlesPosRy), ADR(',"spin":['));
		tmpCalc := ((pShuttleInfo.Position.Ry/17.453293));
		tmpString := REAL_TO_STRING(tmpCalc);
		brdkStrCat(ADR(showShuttlesPosRy), ADR(tmpString));
		brdkStrCat(ADR(showShuttlesPosRy), ADR(',200,2.5'));
		brdkStrCat(ADR(showShuttlesPosRy), ADR(']},'));
		brdkStrCat(ADR(showShuttlesPosRy), ADR('{"select":"#ShuttleTop'));
		brdkStrCat(ADR(showShuttlesPosRy), ADR('","display":'));
		brdkStrCat(ADR(showShuttlesPosRy), ADR('true'));
		brdkStrCat(ADR(showShuttlesPosRy), ADR(',"translate":['));
		tmpCalc := (0);
		tmpString := REAL_TO_STRING(tmpCalc);
		brdkStrCat(ADR(showShuttlesPosRy), ADR(tmpString));
		brdkStrCat(ADR(showShuttlesPosRy), ADR(','));
		tmpCalc := (((pShuttleInfo.Position.Z)*-1)*5);
		tmpString := REAL_TO_STRING(tmpCalc);
		brdkStrCat(ADR(showShuttlesPosRy), ADR(tmpString));
		brdkStrCat(ADR(showShuttlesPosRy), ADR(']'));
		brdkStrCat(ADR(showShuttlesPosRy), ADR(',"spin":['));
		tmpCalc := ((pShuttleInfo.Position.Ry/17.453293));
		tmpString := REAL_TO_STRING(tmpCalc);
		brdkStrCat(ADR(showShuttlesPosRy), ADR(tmpString));
		brdkStrCat(ADR(showShuttlesPosRy), ADR(',200,2.5'));

//		brdkStrCat(ADR(showShuttlesPosRy), ADR(']},'));

		// Select the text
//		brdkStrCat(ADR(showShuttlesPosRy), ADR(TESTString));
//		brdkStrCat(ADR(showShuttlesPosRy), ADR('{"select":"#TextId'));

//		tmpString := USINT_TO_STRING(i+1);
//		brdkStrCat(ADR(showShuttlesPosRy), ADR(tmpString));
//		brdkStrCat(ADR(showShuttlesPosRy), ADR('","display":'));
//		brdkStrCat(ADR(showShuttlesPosRy), ADR('true'));
//		brdkStrCat(ADR(showShuttlesPosRy), ADR('>test</'));

		brdkStrCat(ADR(showShuttlesPosRy), ADR(']}]'));
		sizeOfArray2 := brdkStrLen(ADR(showShuttlesPosRy));

	END_IF

	//showShuttles := '';
	//showShuttles := '[{"select":"#rect1","display":false, "translate":[100,100]}]';
END_ACTION
```

#### Main.st
```iecst
PROGRAM _INIT

	init := TRUE;
	TempTestString := 'Test';

	(*	   <text class="TextID" font-family="Arial" font-size="40" y="70" x="50" font-weight="bold">ID:</text>
	   <text class="TextXY1" font-family="Arial" font-size="25" y="110" x="50" font-weight="bold">X: Y: </text>
	   <text class="TextRxRy1" font-family="Arial" font-size="25" y="150" x="50" font-weight="bold">Rx: Ry: </text>
	   <text class="TextZRz1" font-family="Arial" font-size="25" y="190" x="50" font-weight="bold">Z: Zx:</text>*)

	offsetHeight[0] := 435;
	offsetHeight[1] := 45;
	offsetOut[0] := 475.0;
	offsetOut[1] := 520.0;

	MTLookUpTable_0.Enable := TRUE;
	MTLookUpTable_0.NodeVectorX := offsetHeight;
	MTLookUpTable_0.FcnValues := offsetOut;
	MTLookUpTable_0.NumberOfNodes := 2;

END_PROGRAM

PROGRAM _CYCLIC

//	IF gDemoSystem THEN
//		gShuttleStartupInfo[0].initXPos := 0.1;
//		gShuttleStartupInfo[0].initYPos := 0.1;
//		gShuttleStartupInfo[0].nextStationSelector:= '2';
//		gShuttleStartupInfo[1].initXPos := 0.3;
//		gShuttleStartupInfo[1].initYPos := 0.3;
//		gShuttleStartupInfo[1].nextStationSelector := '3';
//		gDemoSystem := FALSE;
//	END_IF

	IF EDGEPOS(visSelectedShuttle = '#rect1') THEN
		gMain.Par.SelectedIndex := 0;
	ELSIF EDGEPOS(visSelectedShuttle = '#rect2')THEN
		gMain.Par.SelectedIndex := 1;
	ELSIF EDGEPOS(visSelectedShuttle = '#rect3')THEN
		gMain.Par.SelectedIndex := 2;
	ELSIF EDGEPOS(visSelectedShuttle = '#rect4')THEN
		gMain.Par.SelectedIndex := 3;
	END_IF

	// draw Shuttles

	nrOfShuttlesHMI := UINT_TO_USINT(gMain.Status.ShuttlesPresent);
	FOR i := 0 TO 4 DO
		pShuttleInfo ACCESS ADR(gVisShuttle.ShuttleInfoVis[i]);
		drawShuttles;
//		pShuttleStartupInfo ACCESS ADR(gShuttleStartupInfo[i]);
//		drawConfigShuttles;
	END_FOR

//	// draw Motor Segments;
//	FOR i := 0 TO NR_OF_SEGMENTS DO
//		pSegments ACCESS ADR(gSegments[i]);
//		drawMotorSegments;
//	END_FOR

	// harrisb - May 18, 2021 : added to set default demo segments
	// Demo segment Layout (show 4 segments)
	IF gSettings.DemoType THEN
//		demoMotorSegmentLayoutCmd := FALSE;
		FOR i := 0 TO NR_OF_SEGMENTS DO
			IF (i = 0)OR(i = 1)OR(i = 5)OR(i = 6)THEN
				gSegments[i].visible := TRUE;
			ELSE
				gSegments[i].visible := FALSE;
			END_IF
		END_FOR
	ELSIF NOT(gSettings.DemoType) THEN
		FOR i := 0 TO NR_OF_SEGMENTS DO
			IF (i = 0)OR(i = 1)THEN
				gSegments[i].visible := TRUE;
			ELSE
				gSegments[i].visible := FALSE;
			END_IF
		END_FOR
	END_IF

	IF EDGE(gSettings.DemoType) THEN
		showTyleSvg := TRUE;
	END_IF

	// draw Motor Segments;
	FOR i := 0 TO NR_OF_SEGMENTS DO
		pSegments ACCESS ADR(gSegments[i]);
		drawMotorSegments;
	END_FOR

	// Reset segment Layout
	IF resetMotorSegmentLayoutCmd THEN
		resetMotorSegmentLayoutCmd := FALSE;
		FOR i := 0 TO NR_OF_SEGMENTS DO
			gSegments[i].visible := TRUE;
		END_FOR
	END_IF

	// Reset Shuttle Startup Layout
	IF resetShuttleInitLayoutCmd THEN
		resetShuttleInitLayoutCmd := FALSE;
		FOR i := 0 TO NUM_SHUTTLES DO
			gShuttleStartupInfo[i].initXPos := 0.42+0.12*(i);
			gShuttleStartupInfo[i].initYPos := 0.060;
		END_FOR
	END_IF

	// Handle tyle click configuration
	IF this.tableConfigClick THEN
		this.tableConfigClick := FALSE;
		brdkStrRemove(ADR(this.tableConfigString),0,3);
		tmpString := this.tableConfigString;
		this.tableConfigID := STRING_TO_USINT(tmpString);
		this.tableConfigID := this.tableConfigID - 1;
		IF gSegments[this.tableConfigID].visible THEN
			gSegments[this.tableConfigID].visible := FALSE;
		ELSE
			gSegments[this.tableConfigID].visible := TRUE;
		END_IF
	END_IF

	// harrisb - May 21, 2021 : Hide disconnected segments
	FOR i := 0 TO NR_OF_SEGMENTS DO

		CASE i OF

			// allow segment 1 to be ON on its own
			0: IF gSegments[i].visible AND NOT((gSegments[i+1].visible)OR(gSegments[i+5].visible)OR(gSegments[i-5].visible))THEN

				END_IF
			5,10,15,20,25,30,35,40,45: IF gSegments[i].visible AND NOT((gSegments[i+1].visible)OR(gSegments[i+5].visible)OR(gSegments[i-5].visible))THEN
					gSegments[i].visible := FALSE;
				END_IF

			4,9,14,19,24,29,34,39,44,49:	IF gSegments[i].visible AND NOT((gSegments[i-1].visible)OR(gSegments[i+5].visible)OR(gSegments[i-5].visible))THEN
					gSegments[i].visible := FALSE;
				END_IF

			ELSE
				IF gSegments[i].visible AND NOT((gSegments[i+1].visible)OR(gSegments[i-1].visible)OR(gSegments[i+5].visible)OR(gSegments[i-5].visible))THEN
					gSegments[i].visible := FALSE;
				END_IF

		END_CASE;

	END_FOR

	// Handle different svg views on config page
	IF showConfigSvgCmd THEN
		showConfigSvgCmd := FALSE;
		showConfigSvg := TRUE;
		showTyleSvg := FALSE;
		shuttleStartPosSvg := FALSE;
	END_IF

	// Handle different svg views on config page
	IF showTyleSvgCmd THEN
		showTyleSvgCmd := FALSE;
		showTyleSvg := TRUE;
		showConfigSvg := FALSE;
		shuttleStartPosSvg := FALSE;
	END_IF

	// Handle different svg views on config page
	IF shuttleStartPosSvgCmd THEN
		shuttleStartPosSvgCmd := FALSE;
		showTyleSvg := FALSE;
		showConfigSvg := FALSE;
		shuttleStartPosSvg := TRUE;
	END_IF

END_PROGRAM

PROGRAM _EXIT
	(* Insert code here *)

END_PROGRAM
```

### Program Logical/Zone (IEC)

#### Variables.var
```iecst
VAR
	zoneState : UDINT;
	MC_BR_ZoneCreate_Acp6D_0 : MC_BR_ZoneCreate_Acp6D;
	ZonePars : McAcp6DCreateZoneParType;
	MC_BR_ZonePowerOff_Acp6D_0 : MC_BR_ZonePowerOff_Acp6D;
	MC_BR_AsmGetZone_Acp6D_0 : MC_BR_AsmGetZone_Acp6D;
END_VAR
```

#### Cyclic.st
```iecst
PROGRAM _CYCLIC

	CASE zoneState OF

		0:
		// Create Zone
		10:
		//	MC_BR_ZoneCreate_Acp6D_0.Assembly := ;
			MC_BR_ZoneCreate_Acp6D_0.Execute := TRUE;
			MC_BR_ZoneCreate_Acp6D_0.Parameters := ZonePars;

			ZonePars.BottomLeft.X := 0.0;
			ZonePars.BottomLeft.Y := 0.240;
			ZonePars.TopRight.X := 0.240;
			ZonePars.TopRight.Y := 0.240;
		//	ZonePars.Name :='1';
		//	ZonePars.ZoneType;
			zoneState := 0;
		// Power on Zone
		20:
		// Power off Zone
		30:
			MC_BR_ZonePowerOff_Acp6D_0.Zone := ADR(MC_BR_AsmGetZone_Acp6D_0.Zone);
			MC_BR_ZonePowerOff_Acp6D_0.Execute := 	TRUE;
				zoneState := 0;
		// Get Zone Info
		40:
			MC_BR_AsmGetZone_Acp6D_0.Enable := TRUE;
			zoneState := 0;
		//	MC_BR_AsmGetZone_Acp6D_0.Next := ;

	END_CASE

	MC_BR_ZoneCreate_Acp6D_0();
	MC_BR_AsmGetZone_Acp6D_0();
	MC_BR_ZonePowerOff_Acp6D_0();

END_PROGRAM
```

#### Init.st
```iecst
PROGRAM _INIT

	MC_BR_ZoneCreate_Acp6D_0.Assembly := ADR(gAssembly6D_1);
	MC_BR_AsmGetZone_Acp6D_0.Assembly := ADR(gAssembly6D_1);

END_PROGRAM
```

Listed in the project but not available here: Logical/Macro/ResetMacroFubs.st
